Universal Robots PolyScope program: seek_destack_130.urp

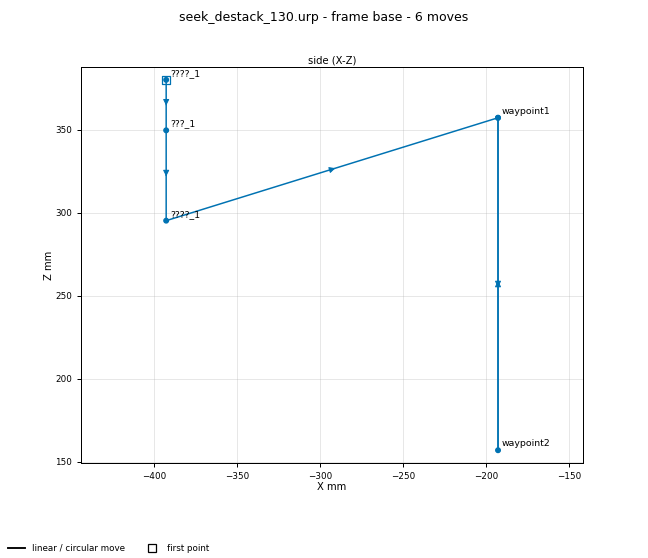
[picture p0: tool path of seek_destack_130.urp in frame base, 6 of 6 moves have a stored position in this frame; points joined in program order, loops and branches not executed]
Program seek_destack_130 (createdIn=3.2.19293 lastSavedIn=3.2.19293 directory=/programs installation=default robotSerialNumber=2015351391)
Calibrated DH parameters: a=[0.000352, -0.161198, -0.373486, 0.00005, 0.000049, 0]; d=[0.089268, 352.477598, -320.08558, -32.281492, 0.094939, 0.082518]; alpha=[1.570728, 0.001116, -0.003686, 1.571189, -1.570572, 0]; deltaTheta=[-0.000012, 1.181849, -1.491165, 0.309495, -0.000007, 0.000025]
Robot Program (runOnlyOnce=false motionType=MoveJ speed=1.047198 acceleration=1.396263 recalculateMotions=false)
  Stack Destack (itemThickness=0.03 motionType=MoveL speed=0.25 acceleration=1.2 recalculateMotions=false) nextPositionExpression=force()>50; foundPoseVariable(name=位姿_1); actionSequence(name=拾取序列 motionType=MoveL speed=0.25 acceleration=1.2 recalculateMotions=false, anchorWaypoint(type=Fixed name=堆垛位置_1, position(joints=2.5762690280602967, -1.674378607626286, -1.6193814247260354, -1.3137377440070512, 1.5891866844234208, -0.26011658411658267 pose=-0.39286558297524965, 0.3789432650022284, 0.38018019540567727, -2.4607974524581966, -1.802590284682575, 0.09027983581124982), poseInFeatureCoordinates=[-0.392866, 0.378943, 0.38018, -2.460797, -1.80259, 0.09028], outputFlangePose=[-0.392876, 0.37892, 0.380185, -2.460705, -1.802665, 0.090452]), feature=Base, children(Waypoint=堆垛位置_1, Set(type=DigitalOutput, pin=Lamp, digitalValue=1), Wait(type=Sleep, waitTime=0.5), Waypoint(type=Fixed name=退出_1, position(joints=2.5762673768156077, -1.6841278825213122, -1.6676683324180868, -1.2557054211529106, 1.5893130504962016, -0.2603042849197914 pose=-0.39288881505343853, 0.3789337731518756, 0.35734681082922964, -2.460629359891928, -1.802699701364262, 0.0905710465662198), poseInFeatureCoordinates=[-0.392889, 0.378934, 0.357347, -2.460629, -1.8027, 0.090571], outputFlangePose=[-0.392876, 0.37892, 0.357366, -2.460705, -1.802665, 0.090452]))); feature=Base
    Waypoint 起始位置_1: TCP in base x=-392.875 y=378.94 z=380.214 mm, rx=-2.4606 ry=-1.8026 rz=0.0904 rad; joints [147.609, -95.935, -92.784, -75.272, 91.054, -14.904] deg
    Direction (stopDistance=0.1 motionType=MoveL speed=0.01 acceleration=1.2 recalculateMotions=false) variable(name=interpolate_1, initializeExpression=0.0); feature=Base
      Waypoint 源位置_1: TCP in base x=-392.875 y=378.937 z=349.789 mm, rx=-2.4608 ry=-1.8027 rz=0.0904 rad; joints [147.609, -96.718, -96.43, -70.843, 91.063, -14.918] deg
      Waypoint 目标位置_1: TCP in base x=-392.874 y=378.947 z=295.344 mm, rx=-2.4605 ry=-1.8026 rz=0.0903 rad; joints [147.609, -98.918, -102.229, -62.844, 91.084, -14.942] deg
    AnchoredSequence -> 拾取序列
  Folder Folder
    MoveL speed 250 mm/s, acceleration 1200 mm/s^2 (recalculateMotions=false) feature=Base
      Waypoint waypoint1: TCP in base x=-192.877 y=378.938 z=357.359 mm, rx=-2.4607 ry=-1.8026 rz=0.0905 rad; joints [131.555, -79.774, -111.525, -73.277, 92.668, -30.878] deg
      Waypoint waypoint2: TCP in base x=-192.859 y=378.941 z=156.968 mm, rx=-2.4608 ry=-1.8028 rz=0.0906 rad; joints [131.557, -95.027, -131.057, -38.499, 92.776, -30.969] deg
      Set DigitalOutput pin=Lamp; digitalValue=0
      Wait Sleep waitTime=0.5
      Waypoint waypoint1: TCP in base x=-192.877 y=378.938 z=357.359 mm, rx=-2.4607 ry=-1.8026 rz=0.0905 rad; joints [131.555, -79.774, -111.525, -73.277, 92.668, -30.878] deg
